// TIA Portal V20 export
TYPE "LConSMC_typeWinderDiag"
// Diagnosedaten des Wicklers / Diagnostic data of the winder
// stored: Access Published
   STRUCT
      typeOfAxis : Int;   // Type of axis 0: Invalid axis 1: Speed axis 2: Positioning axis 3: Synchronous axis
      referenceVelocity : LReal;   // [TO unit] Reference velocity which can be used for an external axis control (winderConfig.axisCtrl = FALSE). Represents the maximum axis velocity at maximum line velocity and minimum diameter
      diameterFactor : LReal;   // [%] Scaling factor for parameter "winderDiag.referenceVelocity" which can be used for an external axis control (winderConfig.axisCtrl = FALSE). Velocity setpoint = referenceVelocity * diameterFactor/100.0. The diameterFactor can directly be copied to the velocityOverride parameter of the TO (<TO>.Override.Velocity)
      diamCalcDiag { S7_SetPoint := 'True'} : "LConSMC_typeDiamCalcDiag";   // Diagnostic structure for diameter calculation
      torquePreControlDiag { S7_SetPoint := 'True'} : "LConSMC_typeTorquePrecontrolDiag";   // Diagnostic structure for torque precontrol
      technologyControllerDiag { S7_SetPoint := 'True'} : "LConSMC_typeTechnollogyControllerDiag";   // Diagnostic structure for technology controller
      webbreakDiag { S7_SetPoint := 'True'} : "LConSMC_typeWebbreakDetectDiag";   // Diagnostic structre for webbreak detection
   END_STRUCT;
END_TYPE
